# EPICS substitutions: db/MicroEpsilon/capaNCDT6500.substitutions
file "capaNCDT6500_chX.template"
{
  pattern { CH_ID,  EGU,  PREC }
          { 1,      "nm", 1    }
          { 2,      "nm", 1    }
          { 3,      "nm", 1    }
          { 4,      "nm", 1    }
          { 5,      "nm", 1    }
          { 6,      "nm", 1    }
          { 7,      "nm", 1    }
          { 8,      "nm", 1    }
}
